                    )
                ]
            ),
            (
                "Transition": "24→0",
                "Condition": "Кнопка \"Комплексное тестирование отключить\"",
                "AlgCondition": "[btn.test_off.out]"
            ),
            (
                "Transition": "N→0",
                "Condition": "Кнопка \"Комплексное тестирование отключить\"",
                "AlgCondition": "[btn.test_off.out]"
            )
        ]
    )
)'}
	testing : T_testing; //Комплексное тестирование
{attribute 'export' := '(
    "type": "TSequence",
    "sequence": (
        "Group": "Блок двигателя",
        "AlgGroup": "bd",
        "Name": "Пуск двигателя",
        "Alg": "[Start_D]",
        "Items": [
            (
                "Transition": "0→1",
                "Condition": "АПК => Пуск двигателя",
                "AlgCondition": "[APK.cmd_start_D]"
            ),
            (
                "Step": "1",
                "Commands": [
                    (
                        "Command": "Открытие крана 11, закрытие крана 10",
                        "AlgCommand": "[cmd_KR11_On]",
                        "Fault": "Кран 11 не открылся, кран 10 не закрылся",
                        "AlgFault": "[am.KR11.notOn OR am.KR10.notOff]"
                    )
                ]
            ),
            (
                "Transition": "1→2",
                "Condition": "Кран 11 открылся, кран 10 закрылся",
                "AlgCondition": "[am.KR11.isOn AND am.KR10.isOff]"
            ),
            (
                "Step": "2",
                "Commands": [
                    (
                        "Command": "Проверка Nтк",
                        "AlgCommand": "[check_Ntk]",
                        "Fault": "Nтк > 100 об/мин",
                        "AlgFault": "[acpar.Ntk.value > 100.0]"
                    )
                ]
            ),
            (
                "Transition": "2→3",
                "Condition": "Nтк < 100 об/мин",
                "AlgCondition": "[acpar.Ntk.value < 100.0]"
            ),
            (
                "Step": "3",
                "Commands": [
                    (
                        "Command": "Открытие крана 12, закрытие крана 9",
                        "AlgCommand": "[cmd_KR12_On]",
                        "Fault": "Кран 12 не открылся, кран 9 не закрылся",
                        "AlgFault": "[am.KR12.notOn OR am.KR9.notOff]"
                    ),
                    (
                        "Command": "Включение Э/М ВНА",
                        "AlgCommand": "[cmd_VNA_On]",
                        "Classifier": "S"
                    ),
                    (
                        "Command": "Открыть КПВ",
                        "AlgCommand": "[cmd_KPV_On]"
                    ),
                    (
                        "Command": "Пуск воздушного стартера",
                        "AlgCommand": "[cmd_VS_On]",
                        "Fault": "Кран 13 не открылся",
                        "AlgFault": "[am.KR13.notOn]"
                    )
                ]
            ),
            (
                "Transition": "3→4",
                "Condition": "Продувка топливного газа",
                "AlgCondition": "[am.KR12.isON AND am.KR9.isOff]"
            ),
            (
                "Step": "4",
                "Commands": [
                    (
                        "Command": "Взвести защиту по ТГ",
                        "AlgCommand": "[cmd_sh_TG_On]"
                    ),
                    (
                        "Command": "СК открыть",
                        "AlgCommand": "[cmd_SK_On]"
                    ),
                    (
                        "Command": "Прокрутка двигателя стартером",
                        "AlgCommand": "[starter_go]"
                    )
                ]
            ),
            (
                "Transition": "4→5",
                "Condition": "Давление ТГ > 20 кгс/см2 И Pm перед ДГ > 15 кгс/см2 И Ntk > 1800 об/мин",
                "AlgCondition": "[aipar.Ptg_inTRK.value > 1.96 AND NOT dipar.Pm_SAR_An.value AND acpar.Ntk.value > 1800]"
            ),
            (
                "Step": "5",
                "Commands": [
                    (
                        "Command": "Открытие крана 15",
                        "AlgCommand": "[am.KR15.on]",
                        "Classifier": "S"
                    ),
                    (
                        "Command": "Взвод защиты по не розжигу на пуске",
                        "AlgCommand": "[cmd_sh_nIgnition]"
                    ),
                    (
                        "Command": "Включение зажигания",
                        "AlgCommand": "[cmd_AZ_On]",
                        "Classifier": "P"
                    ),
                    (
                        "Command": "Пуск двигателя",
                        "AlgCommand": "[FuelReg.fReg.startCom]"
                    )
                ]
            ),
            (
                "Transition": "5→6",
                "Condition": "Nтк > 4500 об/мин",
                "AlgCondition": "[acpar.Ntk.value > 4500]"
            ),
            (
                "Step": "6",
                "Commands": [
                    (
                        "Command": "Взвод защиты по не раскрутке",
                        "AlgCommand": "[cmd_sh_nBoost]",
                        "Classifier": "P"
                    ),
                    (
                        "Command": "Останов воздушного стартера",
                        "AlgCommand": "[cmd_VS_Off]",
                        "Fault": "Кран 13 не закрылся",
                        "AlgFault": "[am.KR13.notOff]"
                    ),
                    (
                        "Command": "Закрытие крана 11, открытие крана 10",
                        "AlgCommand": "[cmd_KR11_Off]",
                        "Fault": "Кран 11 не закрылся, кран 10 не открылся",
                        "AlgFault": "[am.KR11.notOff OR am.KR10.notOn]"
                    ),
                    (
                        "Command": "Кран 15 закрыть",
                        "AlgCommand": "[am.KR15.on]",
                        "Classifier": "R"
                    )
                ]
            ),
            (
                "Transition": "6→7",
                "Condition": "Переход двигателя в режим прогрева",
                "AlgCondition": "[FuelReg.fReg.heating]",
                "DelayTime": "10"
            ),
            (
                "Step": "7",
                "Commands": [
                    (
                        "Command": "Отключение Э/М ВНА",
                        "AlgCommand": "[cmd_VNA_On]",
                        "Classifier": "R"
                    ),
                    (
                        "Command": "Отключение маслонасоса уплотнения",
                        "AlgCommand": "[cmd_PNU_Off]",
                        "Fault": "Маслонасос уплотнений не выключился",
                        "AlgFault": "[am.PNU.notOff]",
                        "Classifier": "P"
                    ),
                    (
                        "Command": "Отключение маслонасоса смазки",
                        "AlgCommand": "[cmd_PNS_Off]",
                        "Fault": "Маслонасос смазки не выключился",
                        "AlgFault": "[am.PNS.notOff]",
                        "Classifier": "P"
                    ),
                    (
                        "Command": "Закрыть КПВ 2, 3, 4",
                        "AlgCommand": "[cmd_KPV234_Off]",
                        "Fault": "КПВ 2, 3, 4 не закрылись",
                        "AlgFault": "[am.KPV2.notOff AND am.KPV3.notOff AND am.KPV4.notOff]",
                        "Classifier": "P"
                    )
                ]
            ),
            (
                "Transition": "7→8",
                "Condition": "Прогрев двигателя",
                "AlgCondition": "[NOT FuelReg.fReg.heating]",
                "DelayTime": "*"
            ),
            (
                "Step": "8",
                "Commands": [
                    (
                        "Command": "Тренирование свечей зажигания",
                        "AlgCommand": "[cmd_AZ_On]",
                        "Classifier": "P"
                    ),
                    (
                        "Command": "Прогрев двигателя окончен",
                        "AlgCommand": "[heating_end]"
                    ),
                    (
                        "Command": "Подъём оборотов",
                        "AlgCommand": "[Ntk_Up]"
                    ),
                    (
                        "Command": "Закрытие КПВ 1, 5",
                        "AlgCommand": "[KPV15_close]",
                        "Fault": "КПВ 1, 5 не закрылись",
                        "AlgFault": "[am.KPV1.notOff AND am.KPV5.notOff]"
                    )
                ]
            ),
            (
                "Transition": "8→9",
                "Condition": "Закрытие КПВ",
                "AlgCondition": "[am.KPV1.isOff AND am.KPV5.isOff]"
            ),
            (
                "Step": "9",
                "Commands": [
                    (
                        "Command": "Завершение",
                        "AlgCommand": "[finish]"
                    )
                ]
            ),
            (
                "Transition": "9→0",
                "Condition": "Логическая 1",
                "AlgCondition": "[TRUE]"
            ),
            (
                "Transition": "N→0",
                "Condition": "Режимы аварийного останова",
                "AlgCondition": "[alg.AO]"
            )
        ]
    )
)'}
	Start_D : T_Start_D; //Пуск двигателя
{attribute 'export' := '(
    "type": "TSequence",
    "sequence": (
        "Group": "Газовая обвязка",
        "AlgGroup": "go",
        "Name": "Заполнение контура компрессора",
        "Alg": "[Filling]",
        "Items": [
            (
                "Transition": "0→1",
                "Condition": "(КПК => Заполнение) ИЛИ (АПК => Заполнение)",
                "AlgCondition": "[KPK.cmd_filling OR APK.cmd_filling]"
            ),
            (
                "Step": "1",
                "Commands": [
                    (
                        "Command": "Кран 4 открыть",
                        "AlgCommand": "[cmd_Kr4_On]",
                        "Fault": "Кран 4 не открылся",
                        "AlgFault": "[am.Kr4.notOn]"
                    )
                ]
            ),
            (
                "Transition": "1→2",
                "Condition": "Кран 4 открыт",
                "AlgCondition": "[am.Kr4.isON]"
            ),
            (
                "Step": "2",
                "Commands": [
                    (
                        "Command": "Продувка контура нагнетателя",
                        "AlgCommand": "[purge]"
                    )
                ]
            ),
            (
                "Transition": "2→3",
                "Condition": "Логическая 1",
                "AlgCondition": "[TRUE]",
                "DelayTime": "10"
            ),
            (
                "Step": "3",
                "Commands": [
                    (
                        "Command": "Кран 5 закрыть",
                        "AlgCommand": "[cmd_Kr5_Off]",
                        "Fault": "Кран 5 не закрылся",
                        "AlgFault": "[am.Kr5.notOff]"
                    )
                ]
            ),
            (
                "Transition": "3→4",
                "Condition": "Кран 5 закрыт",
                "AlgCondition": "[am.Kr5.isOFF]"
            ),
            (
                "Step": "4",
                "Commands": [
                    (
                        "Command": "Заполнение",
                        "AlgCommand": "[filling]",
                        "Fault": "Прирост давления в контуре > 0.05 МПа в секунду ",
                        "AlgFault": "[NOT  alg.nIncPgN]"
                    ),
                    (
                        "Command": "Давление в контуре 30 кгс/см2",
                        "AlgCommand": "[Pg_Ok]",
                        "Fault": "Давление в контуре < 30 кгс/см2",
                        "AlgFault": "[aipar.Pg_outN.value < 2.942]"
                    )
                ]
            ),
            (
                "Transition": "4→5",
                "Condition": "Рост давления в контуре > 0.2 МПа в секунду И давление в контуре > 30 кгс/см2",
                "AlgCondition": "[alg.nIncPgN AND aipar.Pg_outN.value > 2.942]"
            ),
            (
                "Step": "5",
                "Commands": [
                    (
                        "Command": "Стабилизация",
                        "AlgCommand": "[stab]"
                    )
                ]
            ),
            (
                "Transition": "5→6",
                "Condition": "Логическая 1",
                "AlgCondition": "[TRUE]",
                "DelayTime": "20"
            ),
            (
                "Step": "6",
                "Commands": [
                    (
                        "Command": "Кран 1 открыть",
                        "AlgCommand": "[cmd_Kr1_On]",
                        "Fault": "Кран 1 не открылся",
                        "AlgFault": "[am.Kr1.notOn]"
                    ),
                    (
                        "Command": "Кран 6 открыть",
                        "AlgCommand": "[cmd_Kr6_On]",
                        "Fault": "Кран 6 не открылся",
                        "AlgFault": "[am.Kr6.notOn]"
                    )
                ]
            ),
            (
                "Transition": "6→7",
                "Condition": "Кран 1 открыт",
                "AlgCondition": "[am.Kr1.isON]"
            ),
            (
                "Step": "7",
                "Commands": [
                    (
                        "Command": "Кран 4 закрыть",
                        "AlgCommand": "[cmd_Kr4_Off]",
                        "Fault": "Кран 4 не закрылся",
                        "AlgFault": "[am.Kr4.notOff]"
                    )
                ]
            ),
            (
                "Transition": "7→8",
                "Condition": "Кран 4 закрыт",
                "AlgCondition": "[am.Kr4.isOFF]"
            ),
            (
                "Step": "8",
                "Commands": [
                    (
                        "Command": "Завершение",
                        "AlgCommand": "[finish]"
                    )
                ]
            ),
            (
                "Transition": "8→0",
                "Condition": "Логическая 1",
                "AlgCondition": "[TRUE]"
            ),
            (
                "Transition": "N→0",
                "Condition": "Режимы аварийного останова",
                "AlgCondition": "[alg.AO]"
            )
        ]
    )
)'}
	Filling : T_Filling; //Заполнение контура компрессора
{attribute 'export' := '(
    "type": "TSequence",
    "sequence": (
        "Group": "Газовая обвязка",
        "AlgGroup": "go",
        "Name": "Стравливание контура компрессора",
        "Alg": "[Bleeding]",
        "Items": [
            (
                "Transition": "0→1",
                "Condition": "(АОсс => Стравливание) ИЛИ (НОсс => Стравливание) ИЛИ (Стравливание => Стравливание)",
                "AlgCondition": "[AOss.cmd_bleeding OR NOss.cmd_bleeding OR Bleeding_full.cmd_bleeding]"
            ),
            (
                "Step": "1",
                "Commands": [
                    (
                        "Command": "Кран 4 закрыть",
                        "AlgCommand": "[cmd_Kr4_Off]",
                        "Fault": "Кран 4 не закрылся",
                        "AlgFault": "[am.Kr4.notOff]"
                    ),
                    (
                        "Command": "Кран 1 закрыть",
                        "AlgCommand": "[cmd_Kr1_Off]",
                        "Fault": "Кран 1 не закрылся",
                        "AlgFault": "[am.Kr1.notOff]"
                    ),
                    (
                        "Command": "Кран 2 закрыть",
                        "AlgCommand": "[cmd_Kr2_Off]",
                        "Fault": "Кран 2 не закрылся",
                        "AlgFault": "[am.Kr2.notOff]"
                    ),
                    (
                        "Command": "Кран 6 закрыть",
                        "AlgCommand": "[cmd_Kr6_Off]",
                        "Fault": "Кран 6 не закрылся",
                        "AlgFault": "[am.Kr6.notOff]"
                    )
                ]
            ),
            (
                "Transition": "1→2",
                "Condition": "Кран 4 закрыт И Кран 1 закрыт И Кран 2 закрыт И Кран 6 закрыт",
                "AlgCondition": "[am.Kr4.isOFF AND am.Kr1.isOFF AND am.Kr2.isOFF AND am.Kr6.isOFF]"
            ),
            (
                "Step": "2",
                "Commands": [
                    (
                        "Command": "Кран 5 открыть",
                        "AlgCommand": "[cmd_Kr5_On]",
                        "Fault": "Кран 5 не открылся",
                        "AlgFault": "[am.Kr5.notOn]"
                    ),
                    (
                        "Command": "Стравливание",
                        "AlgCommand": "[bleeding]",
                        "Fault": "Р газа на входе К > 0.2 МПа",
                        "AlgFault": "[aipar.Pg_inN.value > 0.2]"
                    )
                ]
            ),
            (
                "Transition": "2→3",
                "Condition": "Кран 5 открыт И Р газа на входе К < 0.2 МПа",
                "AlgCondition": "[am.Kr5.isON AND aipar.Pg_inN.value < 0.2]"
            ),
            (
                "Step": "3",
                "Commands": [
                    (
                        "Command": "Завершение",
                        "AlgCommand": "[finish]"
                    )
                ]
            ),
            (
                "Transition": "3→0",
                "Condition": "Логическая 1",
                "AlgCondition": "[TRUE]"
            ),
            (
                "Transition": "N→0",
                "Condition": "Отсутствие запускающих режимов",
                "AlgCondition": "[NOT mde.NOss AND NOT mde.AOss AND NOT bleeding_full.drm.active]"
            )
        ]
    )
)'}
	Bleeding : T_Bleeding; //Стравливание контура компрессора
END_VAR
(* global variable list subsystem *)
{region INFO}
(*
 Назначение: Статусы подсистем
 Автор:  /Разработчик/ 08.08.2025 8:32:24
 Создано из конфигуратора переменных
*)
{endregion}
{attribute 'qualified_only'}
{attribute 'symbol' := 'read'}
VAR_GLOBAL
	EXT : Tsubsystem := (number := 1); //Подсистема: Внешние источники/№1
	BD : Tsubsystem := (number := 2); //Подсистема: Блок двигателя/№2
	MSD : Tsubsystem := (number := 3); //Подсистема: Маслосистема двигателя/№3
	VS : Tsubsystem := (number := 4); //Подсистема: Воздушный стартер/№4
	AVOM : Tsubsystem := (number := 5); //Подсистема: Аппарат воздушного охлаждения масла двигателя/№5
	BTG : Tsubsystem := (number := 6); //Подсистема: Блок топливного газа/№6
	BPG : Tsubsystem := (number := 7); //Подсистема: Блок пускового газа/№7
	POS : Tsubsystem := (number := 8); //Подсистема: Противообледенительная система и воздухоочистное устройство/№8
	BN : Tsubsystem := (number := 9); //Подсистема: Компрессорная установка/блок нагнетателя/№9
	BU : Tsubsystem := (number := 10); //Подсистема: Блок управления/№10
	GO : Tsubsystem := (number := 11); //Подсистема: Газовая обвязка/№11
	ShC : Tsubsystem := (number := 12); //Подсистема: Контроль защит/№12
END_VAR
    TASK TASK_DIAGN(INTERVAL := T#1000ms, PRIORITY := 10);
    TASK base(INTERVAL := T#200ms, PRIORITY := 3);
    TASK fast(INTERVAL := T#20ms, PRIORITY := 2);
    TASK TASK_TIMESync(INTERVAL := PT2M50.5032704S, PRIORITY := 15);
    TASK Slave104Task(INTERVAL := T#20ms, PRIORITY := 4);
    TASK slow(INTERVAL := T#1000ms, PRIORITY := 5);
    TASK imit(INTERVAL := T#40ms, PRIORITY := 2);
    PROGRAM DIAGN WITH TASK_DIAGN : DIAGN;
    PROGRAM HAND_DIAGN WITH TASK_DIAGN : HAND_DIAGN;
    PROGRAM PRG_base WITH base : PRG_base;
    PROGRAM PRG_PRU_Base WITH base : PRG_PRU_Base;
    PROGRAM PRG_fast WITH fast : PRG_fast;
    PROGRAM PRG_PRU_TimeSync WITH TASK_TIMESync : PRG_PRU_TimeSync;
    PROGRAM _Slave_104_OS.BusTask WITH Slave104Task : _Slave_104_OS.BusTask;
    PROGRAM PRG_slow WITH slow : PRG_slow;
    PROGRAM PRG_IMIT WITH imit : PRG_IMIT;
  END_RESOURCE
END_CONFIGURATION

CONFIGURATION _Slave_104_OS
END_CONFIGURATION

CONFIGURATION UCP1_A1_CU1_RS485
END_CONFIGURATION

CONFIGURATION ModbusSerialSlaveOS_PRU
END_CONFIGURATION

CONFIGURATION Regul_Bus_OS
END_CONFIGURATION

CONFIGURATION UCP1_A1_1
END_CONFIGURATION

CONFIGURATION UCP1_A1_ST1
END_CONFIGURATION

CONFIGURATION UCP1_A1_PP1
END_CONFIGURATION

CONFIGURATION UCP1_A1_CU1
END_CONFIGURATION

CONFIGURATION UCP1_A1_FI1
END_CONFIGURATION

CONFIGURATION UCP1_A1_FI2
END_CONFIGURATION

CONFIGURATION UCP1_A1_AI1
END_CONFIGURATION

CONFIGURATION UCP1_A1_AI2
END_CONFIGURATION

CONFIGURATION UCP1_A1_AI3
END_CONFIGURATION

CONFIGURATION UCP1_A1_AI4
END_CONFIGURATION

CONFIGURATION UCP1_A1_AI5
END_CONFIGURATION

CONFIGURATION UCP1_A1_AI6
END_CONFIGURATION

CONFIGURATION UCP1_A1_AI7
END_CONFIGURATION

CONFIGURATION UCP1_A1_ST2
END_CONFIGURATION

CONFIGURATION UCP1_A2_1
END_CONFIGURATION

CONFIGURATION UCP1_A2_ST1
END_CONFIGURATION

CONFIGURATION UCP1_A2_PP1
END_CONFIGURATION

CONFIGURATION UCP1_A2_AO1
END_CONFIGURATION

CONFIGURATION UCP1_A2_DI1
END_CONFIGURATION

CONFIGURATION UCP1_A2_DI2
END_CONFIGURATION

CONFIGURATION UCP1_A2_DI3
END_CONFIGURATION

CONFIGURATION UCP1_A2_DO1
END_CONFIGURATION

CONFIGURATION UCP1_A2_DI4
END_CONFIGURATION

CONFIGURATION UCP1_A2_ST2
END_CONFIGURATION

CONFIGURATION UE1_A1_1
END_CONFIGURATION

CONFIGURATION UE1_A1_ST1
END_CONFIGURATION

CONFIGURATION UE1_A1_PP1
END_CONFIGURATION

CONFIGURATION UE1_A1_DI1
END_CONFIGURATION

CONFIGURATION UE1_A1_DI2
END_CONFIGURATION

CONFIGURATION UE1_A1_DI3
END_CONFIGURATION

CONFIGURATION UE1_A1_DI4
END_CONFIGURATION

CONFIGURATION UE1_A1_DI5
END_CONFIGURATION

CONFIGURATION UE1_A1_DO1
END_CONFIGURATION

CONFIGURATION UE1_A1_DI6
END_CONFIGURATION

CONFIGURATION UE1_A1_DO2
END_CONFIGURATION

CONFIGURATION UE1_A1_DI7
END_CONFIGURATION

CONFIGURATION UE1_A1_ST2
END_CONFIGURATION

CONFIGURATION UPD1_A1_1
END_CONFIGURATION

CONFIGURATION UPD1_A1_DI1
END_CONFIGURATION

CONFIGURATION UPD1_A1_DI2
END_CONFIGURATION

CONFIGURATION UPD1_A1_DI3
END_CONFIGURATION
